(* Logix 5000 project; controller axis1 vendor 1 type 14 code 155 rev 20.12; software revision 20.01 *)

TASK MainTask (continuous, watchdog 500 ms) : MainProgram

MODULES
   Local : vendor 1 type 14 code 155 (PointIO 0, rev 20.12)
      Kinetix_350 : vendor 1 type 37 code 27 (Ethernet 192.168.1.7, rev 1.1, MotionDiagnostics RPI 1 ms, MotionSync RPI 2 ms)
       : 1734-IE2V (PointIO 2, rev 3.1, Input RPI 80 ms)
      Discrete_IO : Embedded (PointIO 1, rev 20.11, Output RPI 20 ms)
       : 1734-OE2V (PointIO 3, rev 3.1, Output RPI 80 ms)
       : vendor 1 type 109 code 13 (PointIO 4, rev 3.1, Output RPI 80 ms)
END_MODULES

VAR_GLOBAL   (* controller tags *)
   Axis_1 : AXIS_CIP_DRIVE;
   Kinetix_350_Quick_Start : MOTION_GROUP;
END_VAR

PROGRAM MainProgram   (* main routine MainRoutine *)
VAR
   Axis1_Motion : MOTION_INSTRUCTION := (FLAGS := 570425344, DN := 1);
   MOVE_step0 : MOTION_INSTRUCTION;
   MOVE_step1 : MOTION_INSTRUCTION := (FLAGS := 704643072, DN := 1, PC := 1);
   MOVE_step2 : MOTION_INSTRUCTION;
   MOVE_step3 : MOTION_INSTRUCTION;
   MOVE_step4 : MOTION_INSTRUCTION;
   MOVE_step5 : MOTION_INSTRUCTION;
   MOVE_step6 : MOTION_INSTRUCTION;
   MOVE_step7 : MOTION_INSTRUCTION;
   MOVE_step8 : MOTION_INSTRUCTION;
   MOVE_step9 : MOTION_INSTRUCTION;
   one_shot0 : BOOL;
   one_shot1 : BOOL;
   one_shot2 : BOOL;
   one_shot3 : BOOL;
   one_shot_npwr : BOOL;
   one_shot_pwr : BOOL := 1;
   state : INT := 1;
   timer0 : TIMER := (PRE := 1000);
   timer1 : TIMER := (PRE := 1000);
   timer2 : TIMER := (PRE := 1000);
   timer3 : TIMER;
END_VAR

ROUTINE MainRoutine   (* ladder *)
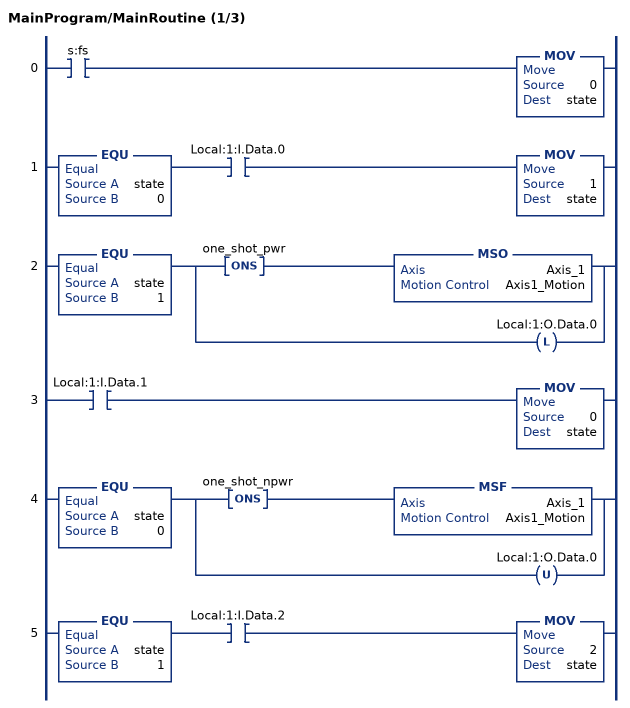
   0: XIC(s:fs)MOV(0,state);
   1: EQU(state,0)XIC(Local:1:I.Data.0)MOV(1,state);
   2: EQU(state,1)[ONS(one_shot_pwr) MSO(Axis_1,Axis1_Motion) ,OTL(Local:1:O.Data.0) ];
   3: XIC(Local:1:I.Data.1)MOV(0,state);
   4: EQU(state,0)[ONS(one_shot_npwr) MSF(Axis_1,Axis1_Motion) ,OTU(Local:1:O.Data.0) ];
   5: EQU(state,1)XIC(Local:1:I.Data.2)MOV(2,state);
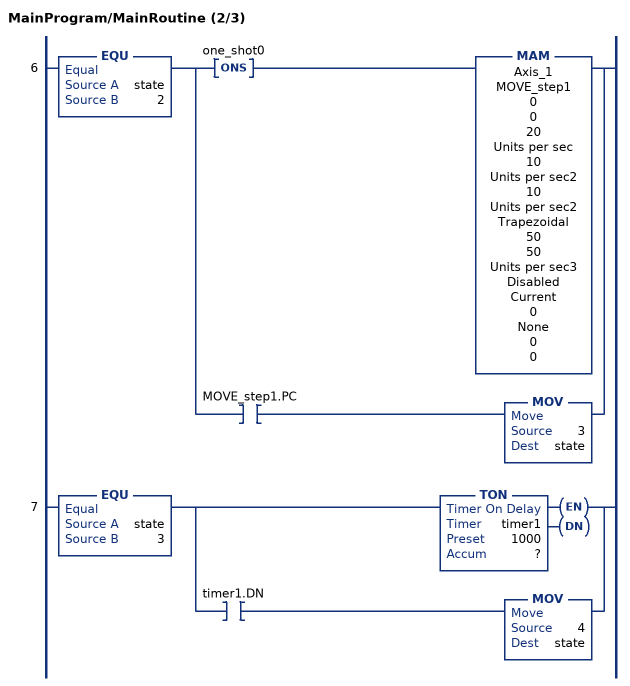
   6: EQU(state,2)[ONS(one_shot0) MAM(Axis_1,MOVE_step1,0,0,20,Units per sec,10,Units per sec2,10,Units per sec2,Trapezoidal,50,50,Units per sec3,Disabled,Current,0,None,0,0) ,XIC(MOVE_step1.PC) MOV(3,state) ];
   7: EQU(state,3)[TON(timer1,?,?) ,XIC(timer1.DN) MOV(4,state) ];
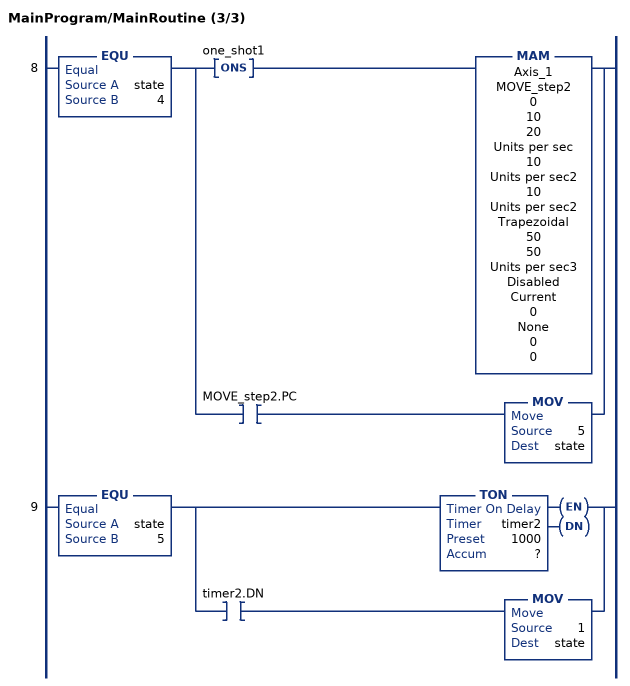
   8: EQU(state,4)[ONS(one_shot1) MAM(Axis_1,MOVE_step2,0,10,20,Units per sec,10,Units per sec2,10,Units per sec2,Trapezoidal,50,50,Units per sec3,Disabled,Current,0,None,0,0) ,XIC(MOVE_step2.PC) MOV(5,state) ];
   9: EQU(state,5)[TON(timer2,?,?) ,XIC(timer2.DN) MOV(1,state) ];
END_ROUTINE
END_PROGRAM
